FUNCTION_BLOCK ValidateFunctionsTest EXTENDS TcUnit.FB_TestSuite
VAR
END_VAR

StringBeginsWithAnyFunction();
StringEndsWithAnyFunction();
StringBeginsWithFunction();
StringEndsWithFunction();

METHOD StringBeginsWithAnyFunction : BOOL
VAR
	test : T_MaxString := 'this is test string';
END_VAR
TcUnit.TEST('String begins with');

AssertEquals_BOOL(
	Expected := FALSE,
	Actual := StringBeginsWithAny(test, 'nothing'),
	Message := 'Should return FALSE because string does not begin with checked value');

AssertEquals_BOOL(
	Expected := TRUE,
	Actual := StringBeginsWithAny(test, 'this'),
	Message := 'Should return TRUE because string begins with checked value');

TEST_FINISHED();
END_METHOD

METHOD StringBeginsWithFunction
VAR
	test : T_MaxString := 'this is test string';
END_VAR
TcUnit.TEST('String begins with Function');

AssertEquals_BOOL(
	Expected := FALSE,
	Actual := StringBeginsWith(test, 'nothing'),
	Message := 'Should return FALSE because string does not begin with checked value');

AssertEquals_BOOL(
	Expected := TRUE,
	Actual := StringBeginsWith(test, 'this'),
	Message := 'Should return TRUE because string begins with checked value');

TEST_FINISHED();
END_METHOD

METHOD StringEndsWithAnyFunction : BOOL
VAR
	test : T_MaxString := 'this is test string';
END_VAR
TcUnit.TEST('String ends with');

AssertEquals_BOOL(
	Expected := FALSE,
	Actual := StringBeginsWithAny(test, 'nothing'),
	Message := 'Should return FALSE because string does not end with checked value');

AssertEquals_BOOL(
	Expected := TRUE,
	Actual := StringEndsWithAny(test, 'string'),
	Message := 'Should return TRUE because string ends with checked value');

TEST_FINISHED();
END_METHOD

METHOD StringEndsWithFunction
VAR
	test : T_MaxString := 'this is test string';
END_VAR
TcUnit.TEST('String ends with Function');

AssertEquals_BOOL(
	Expected := FALSE,
	Actual := StringBeginsWith(test, 'nothing'),
	Message := 'Should return FALSE because string does not end with checked value');

AssertEquals_BOOL(
	Expected := TRUE,
	Actual := StringEndsWith(test, 'string'),
	Message := 'Should return TRUE because string ends with checked value');

TEST_FINISHED();
END_METHOD

END_FUNCTION_BLOCK

(* stored: Version 1.1.0.1, ProductVersion 3.1.4024.12
   POU ValidateFunctionsTest: Id {d8bfc5df-919a-03d7-1337-8a47f04003ad}, SpecialFunc None
   Method StringBeginsWithAnyFunction: Id {e513f70c-a34b-048a-001b-48c3a603580b}
   Method StringBeginsWithFunction: Id {c5106f1a-78ce-0509-007c-c7e3b24fc43b}
   Method StringEndsWithAnyFunction: Id {022e8947-c002-0f07-3f8f-01e15902521a}
   Method StringEndsWithFunction: Id {f4e86b06-ab4c-0da3-339d-d3d3932cf0fc} *)
